(* Logix 5000 project; controller Week_4_PLC_1_Math_Instructions Emulate 5570 rev 30.12; software revision 30.01 *)

TASK MainTask (continuous, watchdog 500 ms) : MainProgram

MODULES
   Local : Emulate 5570 (ICP 2, rev 30.12)
END_MODULES

PROGRAM MainProgram   (* main routine MainRoutine *)
VAR
   Counter : COUNTER := (PRE := 10);
   PB1 : BOOL;
   Value1 : DINT;
   Value2 : DINT;
   Value3 : DINT;
   Value4 : REAL;
END_VAR

ROUTINE MainRoutine   (* ladder *)
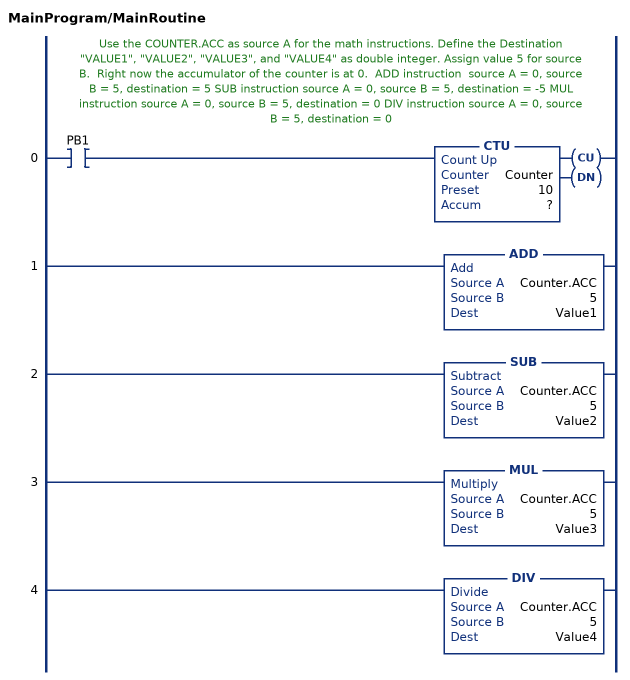
   // Use the COUNTER.ACC as source A for the math instructions. Define the Destination "VALUE1", "VALUE2", "VALUE3", and "VALUE4" as double integer. Assign value 5 for source B.  Right now the accumulator of the counter is at 0.  ADD instruction  source A = 0, source B = 5, destination = 5 SUB instruction source A = 0, source B = 5, destination = -5 MUL instruction source A = 0, source B = 5, destination = 0 DIV instruction source A = 0, source B = 5, destination = 0
   0: XIC(PB1)CTU(Counter,?,?);
   1: ADD(Counter.ACC,5,Value1);
   2: SUB(Counter.ACC,5,Value2);
   3: MUL(Counter.ACC,5,Value3);
   4: DIV(Counter.ACC,5,Value4);
END_ROUTINE
END_PROGRAM
